// Mitsubishi GX Works2 project: counter1   PLC: Q03UDV

PROGRAM MAIN
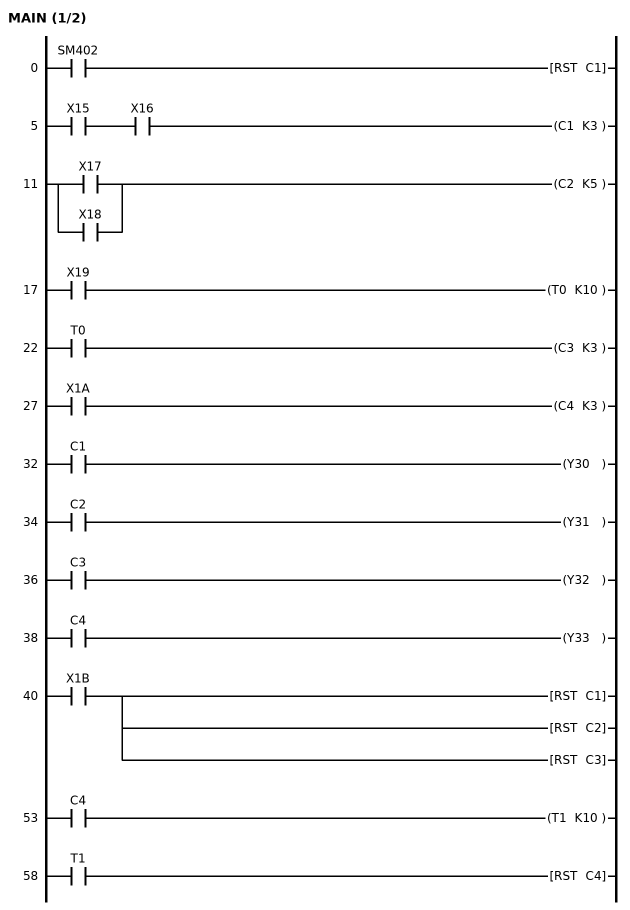
0     LD      SM402
      RST     C1
5     LD      X15
      AND     X16
      OUT     C1 K3
11    LD      X17
      OR      X18
      OUT     C2 K5
17    LD      X19
      OUT     T0 K10
22    LD      T0
      OUT     C3 K3
27    LD      X1A
      OUT     C4 K3
32    LD      C1
      OUT     Y30
34    LD      C2
      OUT     Y31
36    LD      C3
      OUT     Y32
38    LD      C4
      OUT     Y33
40    LD      X1B
      RST     C1
      RST     C2
      RST     C3
53    LD      C4
      OUT     T1 K10
58    LD      T1
      RST     C4
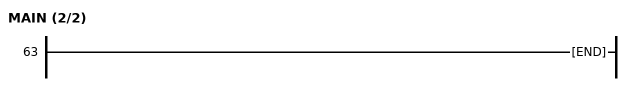
63    END
END_PROGRAM
